FUNCTION F_LogInfo : STRING;
VAR_INPUT
	Message : T_MaxString;
END_VAR

F_LogInfo := F_Logger(ADSLOG_MSGTYPE_HINT, Message);

END_FUNCTION

(* stored: Version 1.1.0.1, ProductVersion 3.1.4020.12
   POU F_LogInfo: Id {a505cbdd-8596-4345-8e8f-adabd9181ab8}, SpecialFunc None *)
